FUNCTION_BLOCK FB_Dynamic_Array
VAR_INPUT
	
END_VAR
VAR_OUTPUT
END_VAR
VAR
	pData 	: POINTER TO T_DATA_TYPE;
	nLength : UDINT;
	t_Null : T_DATA_TYPE;
END_VAR
VAR CONSTANT
	nMIN_UDINT : UDINT := 1;
	nMAX_UDINT : UDINT := 429496729;
END_VAR

(* Get element in array from specified poisiton. *)
METHOD Access : T_DATA_TYPE
VAR_INPUT
	nPosition : UDINT;  // Position of element in dynamic array, 0 indexed.
END_VAR
IF THIS^.Is_Empty() THEN FB_Init(FALSE,FALSE,(nPosition+1)*2); END_IF
IF nPosition >= THIS^.Size() THEN THIS^.Insert(0, nPosition); END_IF
Access := THIS^.pData[nPosition];
END_METHOD

(* Deletes array from memory. *)
METHOD Clear
VAR_INPUT
END_VAR
IF NOT(THIS^.Is_Empty()) THEN __DELETE(THIS^.pData); THIS^.Is_Empty(); END_IF
END_METHOD

METHOD FB_exit : BOOL
VAR_INPUT
	bInCopyCode : BOOL; // if TRUE, the exit method is called for exiting an instance that is copied afterwards (online change).
END_VAR
THIS^.Clear();
END_METHOD

METHOD FB_init : BOOL
VAR_INPUT
	bInitRetains 	: BOOL; 	// if TRUE, the retain variables are initialized (warm start / cold start)
	bInCopyCode 	: BOOL;  	// if TRUE, the instance afterwards gets moved into the copy code (online change)
	nLength 		: UDINT; 	// Length to initialize array with, default is 10;
END_VAR
THIS^.Clear();
IF nLength <> 0 THEN THIS^.pData := __NEW(T_DATA_TYPE, nLength); END_IF
THIS^.nLength := nLength;
END_METHOD

(* Insert element into array at specified position. *)
METHOD Insert
VAR_INPUT
	Data 		: T_DATA_TYPE; 	// Data to insert in dynamic array.
	nPosition 	: UDINT; 		// Position to insert data at in the dynamic array, 0 indexed. 
END_VAR
VAR
	pTemp_Data : POINTER TO T_DATA_TYPE;
	nTemp_Length : UDINT;
	i : DINT;
END_VAR
IF THIS^.Is_Empty() THEN FB_Init(FALSE,FALSE,(nPosition+1)*2); END_IF
IF nPosition < THIS^.Size() THEN 
	THIS^.pData[nPosition] := Data;
ELSE 
	pTemp_Data 		:= THIS^.pData; 
	nTemp_Length 	:= THIS^.nLength;
	THIS^.nLength 	:= (nPosition+1)*2;
	THIS^.pData 	:= __NEW(T_DATA_TYPE, THIS^.nLength);
	FOR i := 0 TO TO_DINT(nTemp_Length-1) DO 
		pData[i] := pTemp_Data[i]; 
		END_FOR
	__DELETE(pTemp_Data);
	THIS^.pData[nPosition] := Data;
	END_IF
END_METHOD

(* Checks if array is empty. *)
METHOD Is_Empty : BOOL
VAR_INPUT
END_VAR
Is_Empty := THIS^.pData = 0;
IF Is_Empty THEN THIS^.nLength := 0; END_IF
END_METHOD

(* Manually resize dynamic array length. If Array become smaller, elements higher positions will be deleted. *)
METHOD Resize
VAR_INPUT
	nLength : UDINT; // New length of dynamic array.
END_VAR
VAR_INST
	pTemp_Data : POINTER TO T_DATA_TYPE;
	nTemp_Length : UDINT;
	i : DINT;
END_VAR
IF nLength = 0 THEN THIS^.Clear(); RETURN; END_IF
IF THIS^.Is_Empty() THEN FB_init(FALSE,FALSE,nLength); RETURN; END_IF
pTemp_Data 		:= THIS^.pData; 
nTemp_Length 	:= THIS^.nLength;
THIS^.nLength 	:= nLength;
THIS^.pData := __NEW(T_DATA_TYPE, THIS^.nLength);
FOR i := 0 TO TO_DINT(nTemp_Length-1) DO 
	IF i > TO_DINT(THIS^.nLength-1) THEN EXIT; END_IF 
	THIS^.pData[i] := pTemp_Data[i]; 
	END_FOR
__DELETE(pTemp_Data);
END_METHOD

(* Display elements in dynamic array in a static array. *)
METHOD Show
VAR_IN_OUT
	aList : ARRAY[*] OF T_DATA_TYPE; // Static array to display data in dynamic array.
END_VAR
VAR
	i,j : DINT; 
END_VAR
FOR i := LOWER_BOUND(aList, 1) TO UPPER_BOUND(aList, 1) DO
	IF (j < TO_DINT(THIS^.Size())) AND NOT(THIS^.Is_Empty()) THEN
		aList[i] := THIS^.pData[j];
		j := j + 1; 
	ELSE 
		aList[i] := t_Null;
	 	END_IF
	END_FOR
END_METHOD

(* Gets the length of dynamic array. *)
METHOD Size : UDINT
VAR_INPUT
END_VAR
Is_Empty(); Size := THIS^.nLength;
END_METHOD

END_FUNCTION_BLOCK

(* stored: Version 1.1.0.1, ProductVersion 3.1.4024.4
   POU FB_Dynamic_Array: Id {151061a5-d3f1-4a43-b5f6-44944bb573cf}, SpecialFunc None
   Method Access: Id {ac0a5f7b-a0d4-4e49-beda-3826bbf28838}
   Method Clear: Id {61bd7724-e2ea-4bde-b7bd-c41ffb9830f3}
   Method FB_exit: Id {ad91c2f7-b680-45b1-adaf-4c5eb0ca9009}
   Method FB_init: Id {ad036e8c-92b0-4824-b55b-41c5ac9fd5d2}
   Method Insert: Id {50f9e499-240c-4146-8b68-b69faf5e63a6}
   Method Is_Empty: Id {1a6f3f50-0bf0-48ce-b0c8-ea0b99aa03ef}
   Method Resize: Id {4bcd3e47-7346-4b8d-8a63-f815ad048ac5}
   Method Show: Id {56bd239f-a051-4f7c-9145-a32b851b5534}
   Method Size: Id {0df4cebf-1354-4f54-bdae-d4b312520a8b} *)
